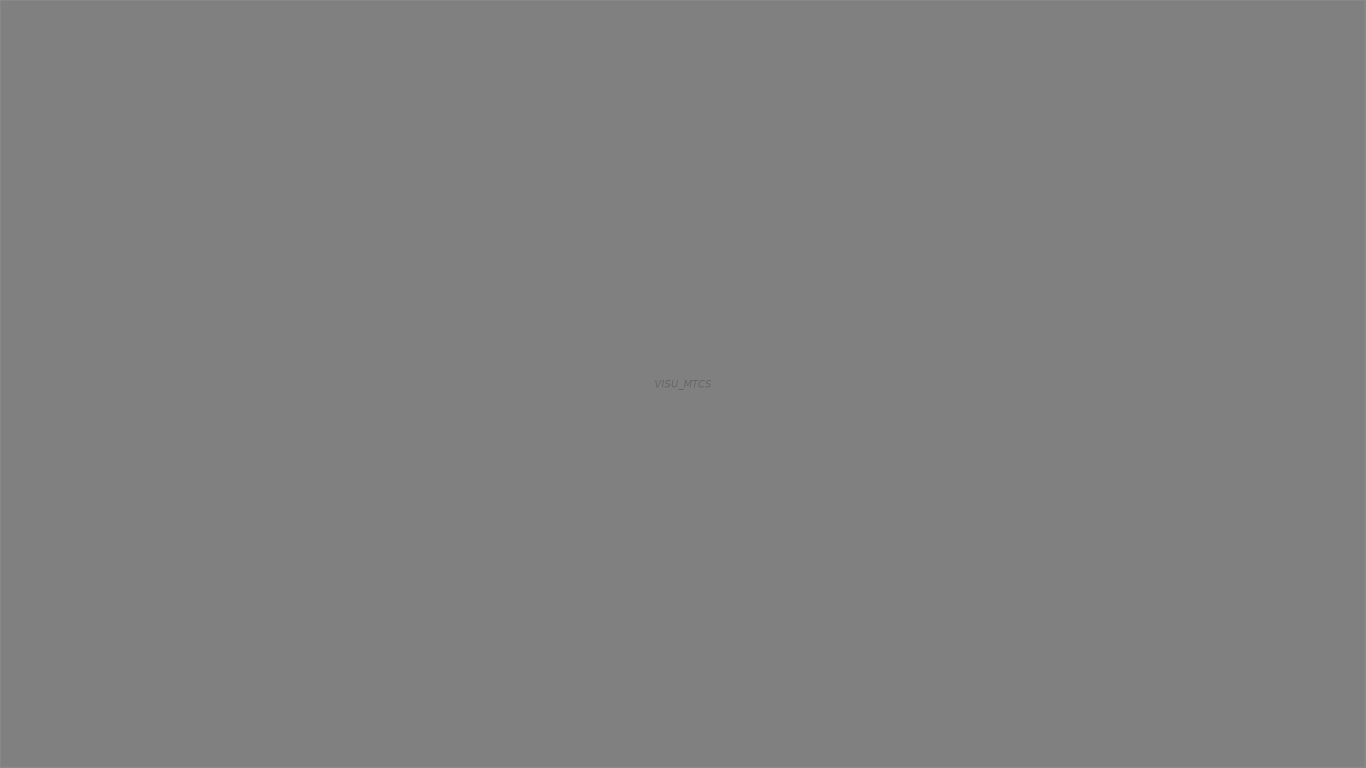
VISUALIZATION VISU_MAIN  // 1366x768
    Frame (0,0 1366x768)
        shows VISU_MTCS(mtcs := GLOBAL.mtcs, mtcsWidget := GLOBAL.gui)
        shows VISU_MTCSBlankScreen(widget := GLOBAL.gui.blankScreen)
END_VISUALIZATION

(* stored: Version 1.1.0.1, ProductVersion 3.1.4019.2
   Visu VISU_MAIN: Id {7a99d089-74b0-4b44-b13c-1c16f276ff98} *)
